TEXTLIST TextList_1Run_1Quartz
  0 = '1 Run = 1 Quartz' | FR: '1 Run = 1 Quartz' | EN: '1 Run = 1 Quartz'
  1 = 'yes' | FR: 'Activé' | EN: 'Activated'
  2 = 'no' | FR: 'Désactivé' | EN: 'Disabled'
  3 = 'raz' | FR: 'Forcage changement quartz' | EN: 'Quartz change forcing'
  4 = 'next' | FR: 'Quartz prévu pour le prochain run' | EN: 'Scheduled quartz for next run'
  5 = 'change' | FR: 'Changement de tous les quartz\n\nnécessaire pour le prochain run' | EN: 'Change all quartz is needed\n\nfor next run'
   = ''
END_TEXTLIST

(* stored: Version 1.1.0.1, ProductVersion 3.1.4024.12
   TextList TextList_1Run_1Quartz: Id {599755ab-b487-48ed-ac1b-951c047c47ca} *)
